// Raw terminal representation. The application owns hardware mapping.
TYPE U_IoRaw_Out :
UNION
    dw    : DWORD;
    fReal : REAL;
    w     : WORD;
    nInt  : INT;
    ui    : UINT;
    di    : DINT;
    udi   : UDINT;
END_UNION
END_TYPE

(* stored: Version 1.1.0.1, ProductVersion 3.1.4026.12
   DUT U_IoRaw_Out: Id {c0000030-0000-0000-0000-000000000004} *)
